// TIA Portal V20 export
FUNCTION_BLOCK "FB_AnalogOutputs"   // FB225, SCL
{ S7_Optimized_Access := 'TRUE' }
// stored: AutoNumber false, MemoryReserve 100, SetENOAutomatically false
   VAR
      sNozzleOverpressureSetPoint { S7_SetPoint := 'True'} : "FB_AnalogOutput";
      sFreeQW482 { S7_SetPoint := 'True'} : "FB_AnalogOutput";
      sVentilatorSetPoint { S7_SetPoint := 'True'} : "FB_AnalogOutput";
      sPropValveClimSetPoint { S7_SetPoint := 'True'} : "FB_AnalogOutput";
   END_VAR
BEGIN
   REGION Description head
       //==================================================================================
       // POSALUX Swiss SA / (C) Copyright 2025
       //----------------------------------------------------------------------------------
       // Title: Analog output function
       // Comment/Function: Analog Ouputs mapping
       // Author: Fabien WALDT
       // Engineering: TIA Portal v17
       //----------------------------------------------------------------------------------
       // Change log table:
       // Version  | Date     | Expert in charge | Changes applied
       // ---------|----------|------------------|-----------------------------------------
       // 00.00.01 | 20250423 | WFA              | First released version
       // =================================================================================
   END_REGION

   // ET200SP Mapping
   REGION IW428 - IW434 : AQ 4xU/I ST Slot 22
       #sNozzleOverpressureSetPoint(iLimitUp := 10.0,
                                    iLimitDown := 0.0,
                                    iMaxAIWordValue := 27648.0,
                                    oValueHW => "AQ_NozzleOverpressureSetPoint");

       #sFreeQW482(iLimitUp := 100.0,
                   iLimitDown := 0.0,
                   iMaxAIWordValue := 27648.0,
                   oValueHW => "AQ_FreeQW482");

       #sVentilatorSetPoint(iLimitUp := 100.0,
                            iLimitDown := 0.0,
                            iMaxAIWordValue := 27648.0,
                            oValueHW => "AQ_VentilatorSetPoint");

       #sPropValveClimSetPoint(iLimitUp := 100.0,
                               iLimitDown := 0.0,
                               iMaxAIWordValue := 27648.0,
                               oValueHW => "AQ_PropValveClimSetPoint");
   END_REGION
END_FUNCTION_BLOCK
